PROGRAM MAIN
VAR
	Eventbuffer: FB_EventBuffer;
	
	AddEvent: BOOL;
	stEventToAdd: ST_Event;
	bEventToAddError: BOOL;
	
	
ReadAndRemoveEvent: BOOL;
stLastReadEvent: ST_Event;

bReadAndRemoveEventError:BOOL;
	nCount: UDINT;
	 
END_VAR

IF AddEvent THEN
	Eventbuffer.AddEvent(stEvent:=stEventToAdd, bError=> bEventToAddError, nCount=> nCount);
	AddEvent:= FALSE;
	
END_IF

IF ReadAndRemoveEvent THEN
		Eventbuffer.GetAndRemoveEvent(stEvent=>stLastReadEvent, bError=> bReadAndRemoveEventError, nCount=> nCount);
ReadAndRemoveEvent:=FALSE;
END_IF

IF StartNotePad THEN
	notepadStart(c
END_IF

END_PROGRAM

(* stored: Version 1.1.0.1, ProductVersion 3.1.4024.11
   POU MAIN: Id {070908f0-aa76-465d-b778-6ce3b20b7726}, SpecialFunc None *)
